PROGRAM MAIN
VAR
	r1:LREAL:=20;
    fbSample : FB_Sample; 
    sMyPath : STRING; 
	teste:FB_Teste;
	grupo:FB_GroupDiag;
END_VAR

safetyDiag();
fbSample(); 
sMyPath := fbSample.sPath;

END_PROGRAM

(* stored: Version 1.1.0.1, ProductVersion 3.1.4024.12
   POU MAIN: Id {f714639e-05df-4447-a78a-06a7cf813137}, SpecialFunc None *)
